INTERFACE ITF_ControlElement6 EXTENDS ITF_BaseControlElement

END_INTERFACE

(* stored: Version 1.1.0.1, ProductVersion 3.1.4024.15
   Itf ITF_ControlElement6: Id {6eadfbc1-2232-4b1b-b5eb-8fe359ff5c6a} *)
